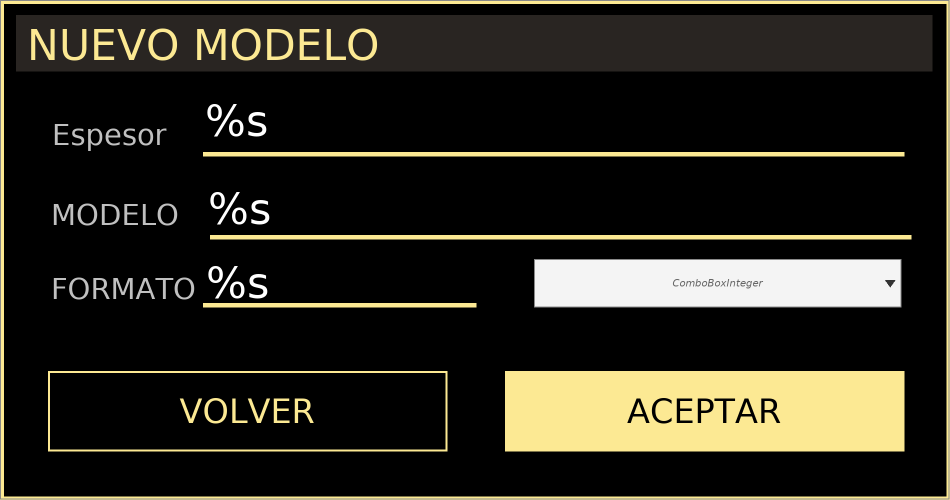
VISUALIZATION Modelo_Tabla_Ch2  // 950x500
    Rectangle (16,15 916x56)
    Rectangle (0,0 950x500)
    Label (24,17 498x56), "NUEVO MODELO"
    Rectangle (136,1125 690x58), "%s Contador piezas corte húmedo 4", text variable: FuncParoNodoRemote1CorteH2.Funci_CortHum2.Min_Parado_Ftc
    Button (871,1105 269x91), "Reset contador"
        tap FuncParoNodoRemote1CorteH2.Funci_CortHum2.ResetContPiez
    ComboBoxInteger (534,259 367x48), variable: FuncParoNodoRemote1CorteH2.FunGeneCortHum2.IndexListFormatoTabla, text list: 'FormatoTabla'
        p1601986498: ''
    Rectangle (205,185 701x48), "%s", text variable: FuncParoNodoRemote1CorteH2.FunGeneCortHum2.s_ModeloEleccionTabla
        OnMouseDown: write the text variable via Edit
    Label (48,197 148x36), "MODELO"
    Rectangle (210,235 701x4)
    Group (48,259 428x48), text variable: FuncParoNodoRemote1CorteH2.FunGeneCortHum2.s_FormatoEleccionTabla, input disabled if: FuncParoNodoRemote1CorteH2.FunGeneCortHum2.IndexListFormatoTabla<>6
        OnMouseClick: write the text variable via Edit
        Rectangle (155,0 273x48), "%s", text variable: FuncParoNodoRemote1CorteH2.sFormatoActualTabla
            OnMouseDown: write the text variable via Edit
        Label (0,12 148x36), "FORMATO"
        Rectangle (155,44 273x4)
    Rectangle (505,371 399x80), "ACEPTAR"
        tap FuncParoNodoRemote1CorteH2.FunGeneCortHum2.P_EscribirModelo
        OnMouseClick: CloseDialog Dialog=Modelo_Tabla_Ch2, Result=OK, NumpadKeypadSet=True
    Rectangle (48,371 399x80), "VOLVER"
        OnMouseClick: CloseDialog Dialog=Modelo_Tabla_Ch2, Result=None, NumpadKeypadSet=True
    Label (49,117 148x36), "Espesor"
    Rectangle (203,152 701x4)
    Rectangle (202,97 701x48), "%s", text variable: FuncParoNodoRemote1CorteH2.FunGeneCortHum2.s_EspesorEleccionTabla
        OnMouseDown: write the text variable via Edit
END_VISUALIZATION

(* stored: Version 1.1.0.1, ProductVersion 3.1.4024.12
   Visu Modelo_Tabla_Ch2: Id {80a4b618-84b7-4e17-b8f6-ff374c3b94b8} *)
